FUNCTION_BLOCK skLoad (* Composite Function Block Type *)
  (* Standard: 61499-2 *)
  (* Version 0.0, 11/8/2025, codex, template *)
  PACKAGE Main;
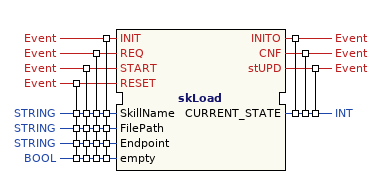
  EVENT_INPUT
    INIT WITH SkillName, FilePath, Endpoint, empty; (* Initialization Request *)
    REQ WITH SkillName, FilePath, Endpoint, empty; (* Normal Execution Request *)
    START WITH SkillName, FilePath, Endpoint, empty;
    RESET WITH SkillName, FilePath, Endpoint, empty;
  END_EVENT
  EVENT_OUTPUT
    INITO WITH CURRENT_STATE; (* Initialization Confirm *)
    CNF WITH CURRENT_STATE; (* Execution Confirmation *)
    stUPD WITH CURRENT_STATE;
  END_EVENT
  VAR_INPUT
    SkillName : STRING;
    FilePath : STRING;
    Endpoint : STRING;
    empty : BOOL;
  END_VAR
  VAR_OUTPUT
    CURRENT_STATE : INT;
  END_VAR
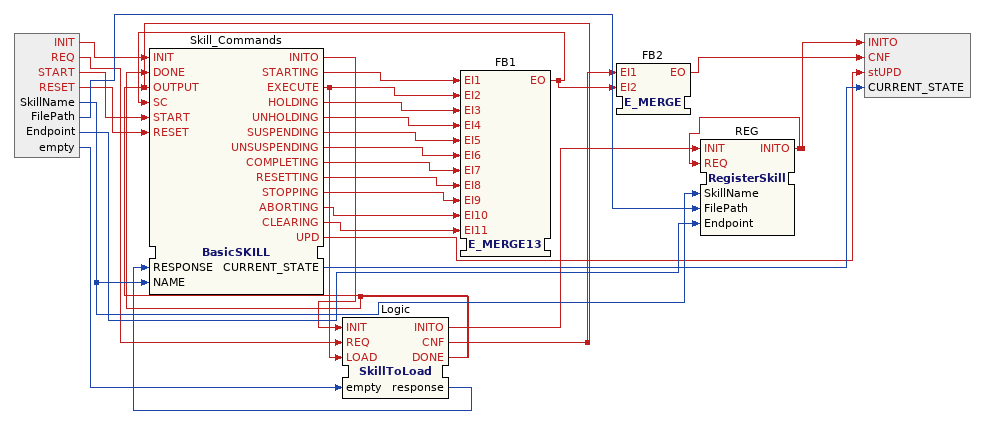
  FBS
    Skill_Commands : BasicSKILL;
    REG : RegisterSkill;
    Logic : SkillToLoad;
    FB1 : E_MERGE13;
    FB2 : E_MERGE;
  END_FBS
  EVENT_CONNECTIONS
    INIT TO Skill_Commands.INIT;
    Skill_Commands.INITO TO Logic.INIT;
    Logic.INITO TO REG.INIT;
    REG.INITO TO REG.REQ;
    REQ TO Logic.REQ;
    REG.INITO TO INITO;
    Skill_Commands.STARTING TO FB1.EI1;
    Skill_Commands.EXECUTE TO Logic.LOAD;
    Skill_Commands.EXECUTE TO FB1.EI2;
    Skill_Commands.HOLDING TO FB1.EI3;
    Skill_Commands.UNHOLDING TO FB1.EI4;
    Skill_Commands.SUSPENDING TO FB1.EI5;
    Skill_Commands.UNSUSPENDING TO FB1.EI6;
    Skill_Commands.COMPLETING TO FB1.EI7;
    Skill_Commands.RESETTING TO FB1.EI8;
    Skill_Commands.STOPPING TO FB1.EI9;
    Skill_Commands.ABORTING TO FB1.EI10;
    Skill_Commands.CLEARING TO FB1.EI11;
    Logic.CNF TO FB2.EI1;
    Logic.DONE TO Skill_Commands.DONE;
    Logic.DONE TO Skill_Commands.OUTPUT;
    FB2.EO TO CNF;
    FB1.EO TO Skill_Commands.SC;
    START TO Skill_Commands.START;
    RESET TO Skill_Commands.RESET;
    Skill_Commands.UPD TO stUPD;
    FB1.EO TO FB2.EI2;
    Logic.CNF TO Skill_Commands.OUTPUT;
  END_CONNECTIONS
  DATA_CONNECTIONS
    SkillName TO REG.SkillName;
    FilePath TO REG.FilePath;
    Endpoint TO REG.Endpoint;
    Logic.response TO Skill_Commands.RESPONSE;
    empty TO Logic.empty;
    SkillName TO Skill_Commands.NAME;
    Skill_Commands.CURRENT_STATE TO CURRENT_STATE;
  END_CONNECTIONS
END_FUNCTION_BLOCK
